PROGRAM PLC_PRG
VAR
//triggers
	trigA0_DI1: R_TRIG;	//trigger for cylinder sensor 

	trigStart: R_TRIG;
END_VAR

//sytem OK
gvl.systemOK := IO.A1_DI0; 
// triggers
trigA0_DI1(clk := IO.A1_DI1);
trigStart (clk := gvl.StartStop); 

IF NOT gvl.systemOK THEN 
	gvl.motor1.en := FALSE; 	//stopping the motors 
	gvl.motor2.en := FALSE;
	
	gvl.StartStop := false; 	//stopping proces
END_IF

//calling program 
automat_PRG(SFCInit := trigStart.Q);

END_PROGRAM

(* stored: Version 1.1.0.1, ProductVersion 3.1.4024.12
   POU PLC_PRG: Id {64ce7901-a7f8-405d-aca1-10be90b183a4}, SpecialFunc None *)
